// TIA Portal V17 export
// export: Created 2025-03-12T14:52:43.107896Z, ExportSetting WithDefaults, DisplayName Totally Integrated Automation Portal, DisplayVersion V17 Update 8, DisplayName TIA Portal Openness, DisplayVersion V17 Update 8, DisplayName TIA Portal Version Control Interface, DisplayVersion V17, DisplayName SINAMICS Startdrive Advanced, DisplayVersion V17 SP2, DisplayName SINAMICS Startdrive G110M, G120, G120C, G120D, G120P, G115D, DisplayVersion V17 SP2, DisplayName SINAMICS Startdrive G130, G150, S120, S150, SINAMICS MV, S210, DisplayVersion V17 SP2, DisplayName STEP 7 Professional, DisplayVersion V17 Update 8, DisplayName SINUMERIK ONE STEP 7 Toolbox, DisplayVersion V17 Update 12, DisplayName SINUMERIK 840D sl STEP 7 Toolbox, DisplayVersion V17 Update 12, DisplayName STEP 7 Safety, DisplayVersion V17 Update 6, DisplayName WinCC Advanced, DisplayVersion V17 Update 8
TYPE "POWDER_FEEDER_LINE"
// stored: IsFailsafeCompliant false
   STRUCT
      HOPPER : Struct
         PRESSURE : Real;   // POWDER FEEDER HOPPER PRESSURE VALUE (Bar)
         TEMPERATURE : Real;   // POWDER FEEDER HOPPER TEMPERATURE VALUE (ºC)
         TEMPERATURE_SETPOINT : Real;   // POWDER FEEDER HOPPER TEMPERATURE SETPOINT VALUE (ºC)
         STIRRER_CURRENT : Int;   // POWDER FEEDER HOPPER STIRRER CURREN VALUE (mA)
         STIRRER_SPEED : Real;   // POWDER FEEDER HOPPER STIRRER SPEED VALUE (RPM or %)
         STIRRER_SPEED_SETPOINT : Real;   // POWDER FEEDER HOPPER STIRRER SPEED SETPOINT VALUE (RPM or %)
      END_STRUCT;
      DISC : Struct
         CURRENT : Int;   // POWDER FEEDER DISC CURRENT VALUE (mA)
         SPEED : Real;   // POWDER FEEDER DISC SPEED VALUE (RPM or %)
         SPEED_SETPOINT : Real;   // POWDER FEEDER DISC SPEED SET POINT VALUE (RPM or %)
      END_STRUCT;
      CARRIER_GAS : Struct
         PRESSURE : Real;   // POWDER FEEDER CARRIER GAS PRESSURE VALUE (Bar)
         FLOW : Real;   // POWDER FEEDER CARRIER GAS FLOW VALUE (NLPM)
         FLOW_SETPOINT : Real;   // POWDER FEEDER CARRIER GAS FLOW SETPOINT VALUE (NLPM)
      END_STRUCT;
      POWDER_FLOW : Array[1..20] of "MEDICOAT_TIME_STAMP";   // POWDER FEEDER POWDER FLOW VALUE (Raw)
      POWDER_TYPE { ExternalWritable := 'False'} : Struct
         MANUFACTURER { ExternalWritable := 'False'} : Array[0..20] of Char;   // POWDER TYPE: MANUFACTURER IDENTIFICATION
         REFERENCE { ExternalWritable := 'False'} : Array[0..20] of Char;   // POWDER TYPE: POWDER REFERENCE
         BATCH_NUMBER { ExternalWritable := 'False'} : Array[0..20] of Char;   // POWDER TYPE: POWDER BATCH NUMBER
         CONTAINER_ID { ExternalWritable := 'False'} : Array[0..20] of Char;   // POWDER TYPE: POWDER CONTAINER IDENTIFICATION
         HUMIDITY { ExternalWritable := 'False'} : Real;   // POWDER TYPE: HUMIDITY VALUE (¿?¿?¿?¿?)
         GRANULOMETRY { ExternalWritable := 'False'} : Real;   // POWDER TYPE: GRANULOMETRY VALUE (¿?¿?¿?¿?)
         POROSITY { ExternalWritable := 'False'} : Real;   // POWDER TYPE: POROSITY VALUE (¿?¿?¿?¿?)
      END_STRUCT;
      STATUS : Struct
         RUNNING : Bool;
      END_STRUCT;
   END_STRUCT;
END_TYPE
